// TIA Portal V20 export
VAR_GLOBAL   // PLC tag table "3.Entrada Analoga"
   Input_analog_1 AT %IW10 : Int;
   Input_analog_2 AT %IW12 : Int;
   Input_analog_3 AT %IW14 : Int;
   Input_analog_4 AT %IW16 : Int;
END_VAR
